FUNCTION_BLOCK changeEventProcess1 (* Basic Function Block Type *)
  (* Standard: 61499-2 *)
  (* Version 0.0, 5/23/2025, azam_w, Schneider Electric, Template *)
  PACKAGE Main;
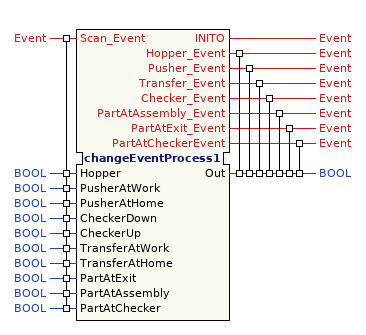
  EVENT_INPUT
    Scan_Event WITH Hopper, PusherAtWork, PusherAtHome, CheckerDown, CheckerUp, TransferAtWork, TransferAtHome, PartAtExit, PartAtAssembly, PartAtChecker;
  END_EVENT
  EVENT_OUTPUT
    INITO; (* Initialization Confirm *)
    Hopper_Event WITH Out; (* Execution Confirmation *)
    Pusher_Event WITH Out;
    Transfer_Event WITH Out;
    Checker_Event WITH Out;
    PartAtAssembly_Event WITH Out;
    PartAtExit_Event WITH Out;
    PartAtCheckerEvent WITH Out;
  END_EVENT
  VAR_INPUT
    Hopper : BOOL; (* Output event qualifier *)
    PusherAtWork : BOOL;
    PusherAtHome : BOOL;
    CheckerDown : BOOL;
    CheckerUp : BOOL;
    TransferAtWork : BOOL;
    TransferAtHome : BOOL;
    PartAtExit : BOOL;
    PartAtAssembly : BOOL;
    PartAtChecker : BOOL;
  END_VAR
  VAR_OUTPUT
    Out : BOOL;
  END_VAR
  VAR
    Hopper_PrevVAl : BOOL := FALSE;
    PusherAtWork_PrevVal : BOOL := FALSE;
    PusherAtHome_PrevVal : BOOL := FALSE;
    TransferAtWork_PrevVal : BOOL := FALSE;
    TransferAtHome_PrevVal : BOOL := FALSE;
    CheckerDown_PrevVal : BOOL := FALSE;
    CheckerUp_PrevVal : BOOL;
    PartAtAssembly_PreVal : BOOL;
    PartAtExit_PreVal : BOOL;
    PartAtChecker_PreVal : BOOL;
  END_VAR
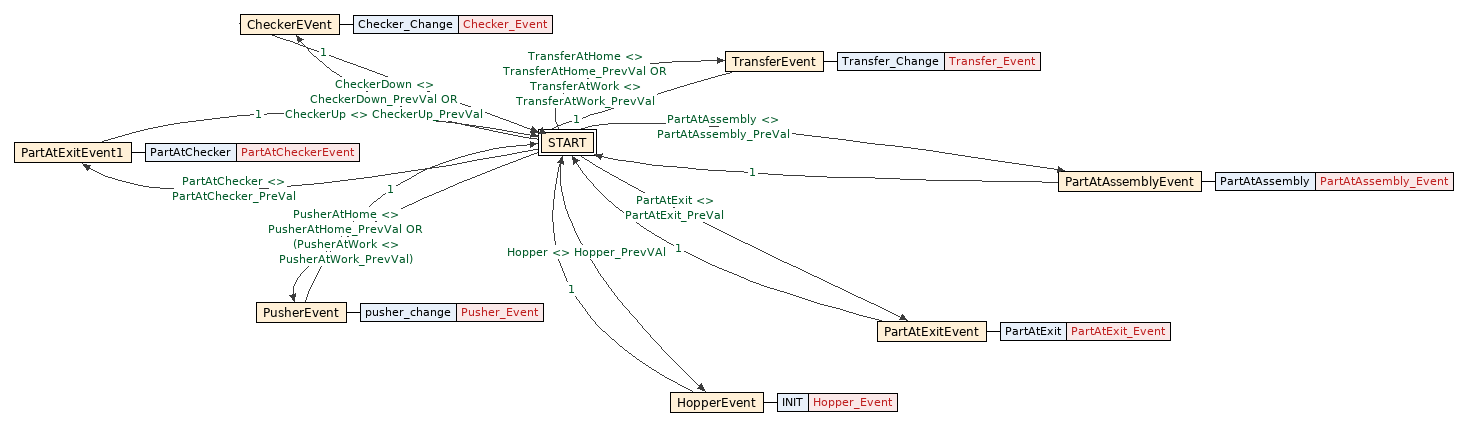
  EC_STATES
    START; (* Initial State *)
    HopperEvent : INIT -> Hopper_Event; (* Normal execution *)
    PusherEvent : pusher_change -> Pusher_Event;
    TransferEvent : Transfer_Change -> Transfer_Event;
    CheckerEVent : Checker_Change -> Checker_Event;
    PartAtAssemblyEvent : PartAtAssembly -> PartAtAssembly_Event; (* Normal execution *)
    PartAtExitEvent : PartAtExit -> PartAtExit_Event; (* Normal execution *)
    PartAtExitEvent1 : PartAtChecker -> PartAtCheckerEvent; (* Normal execution *)
  END_STATES
  EC_TRANSITIONS
    START TO HopperEvent := Hopper <> Hopper_PrevVAl;
    HopperEvent TO START := 1;
    START TO PusherEvent := PusherAtHome <> PusherAtHome_PrevVal OR (PusherAtWork <> PusherAtWork_PrevVal);
    PusherEvent TO START := 1;
    START TO TransferEvent := TransferAtHome <> TransferAtHome_PrevVal OR TransferAtWork <> TransferAtWork_PrevVal;
    TransferEvent TO START := 1;
    START TO CheckerEVent := CheckerDown <> CheckerDown_PrevVal OR CheckerUp <> CheckerUp_PrevVal;
    CheckerEVent TO START := 1;
    START TO PartAtAssemblyEvent := PartAtAssembly <> PartAtAssembly_PreVal;
    PartAtAssemblyEvent TO START := 1;
    START TO PartAtExitEvent := PartAtExit <> PartAtExit_PreVal;
    PartAtExitEvent TO START := 1;
    START TO PartAtExitEvent1 := PartAtChecker <> PartAtChecker_PreVal;
    PartAtExitEvent1 TO START := 1;
  END_TRANSITIONS
  ALGORITHM INIT IN ST: (* Initialization algorithm *)
;
IF Hopper <> Hopper_PrevVAl THEN
	Hopper_PrevVAl := Hopper;
	Out := Hopper;
END_IF;
  END_ALGORITHM
  ALGORITHM REQ IN ST: (* Normally executed algorithm *)
;

IF Hopper <> Hopper_PrevVAl THEN
	Hopper_PrevVAl := Hopper;
    Out := Hopper;
END_IF;
  END_ALGORITHM
  ALGORITHM pusher_change IN ST:
;

IF PusherAtWork <> PusherAtWork_PrevVal THEN
	PusherAtWork_PrevVal := PusherAtWork;
	Out := PusherAtWork;
END_IF;

IF PusherAtHome <> PusherAtHome_PrevVal THEN
	PusherAtHome_PrevVal := PusherAtHome;
	Out := PusherAtHome;
END_IF;
  END_ALGORITHM
  ALGORITHM Transfer_Change IN ST:
;

IF TransferAtHome <> TransferAtHome_PrevVal THEN
	TransferAtHome_PrevVal := TransferAtHome;
	Out := TransferAtHome;
END_IF;

IF TransferAtWork <> TransferAtWork_PrevVal THEN
	TransferAtWork_PrevVal := TransferAtWork;
	Out := TransferAtWork;
END_IF;
  END_ALGORITHM
  ALGORITHM Checker_Change IN ST:
;

IF CheckerDown <> CheckerDown_PrevVal THEN
	CheckerDown_PrevVal := CheckerDown;
	Out := CheckerDown;
END_IF;

IF CheckerUp <> CheckerUp_PrevVal THEN
	CheckerUp_PrevVal := CheckerUp;
	Out := CheckerUp;
END_IF;
  END_ALGORITHM
  ALGORITHM PartAtAssembly IN ST:
;
IF PartAtAssembly <> PartAtAssembly_PreVal THEN
	PartAtAssembly_PreVal := PartAtAssembly;
	Out := PartAtAssembly;
END_IF;
  END_ALGORITHM
  ALGORITHM PartAtExit IN ST:
;
 IF PartAtExit <> PartAtExit_PreVal THEN
	PartAtExit_PreVal := PartAtExit;
	Out := PartAtExit;
END_IF;
  END_ALGORITHM
  ALGORITHM PartAtChecker IN ST:
;
 IF PartAtChecker <> PartAtChecker_PreVal THEN
	PartAtChecker_PreVal := PartAtChecker;
	Out := PartAtChecker;
END_IF;
  END_ALGORITHM
END_FUNCTION_BLOCK
